FUNCTION_BLOCK CallButtons (* Composite Function Block Type *)
  (* Standard: 61499-2 *)
  (* Version 0.0, 11/8/2016, Dmitry, nxtControl GmbH, template *)
  PACKAGE Main;
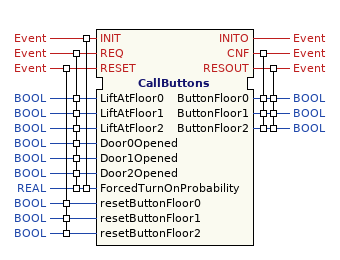
  EVENT_INPUT
    INIT WITH ForcedTurnOnProbability; (* Initialization Request *)
    REQ WITH LiftAtFloor0, LiftAtFloor1, LiftAtFloor2, Door0Opened, Door1Opened, Door2Opened, ForcedTurnOnProbability; (* Normal Execution Request *)
    RESET WITH resetButtonFloor0, resetButtonFloor1, resetButtonFloor2;
  END_EVENT
  EVENT_OUTPUT
    INITO; (* Initialization Confirm *)
    CNF WITH ButtonFloor0, ButtonFloor1, ButtonFloor2; (* Execution Confirmation *)
    RESOUT WITH ButtonFloor0, ButtonFloor1, ButtonFloor2;
  END_EVENT
  VAR_INPUT
    LiftAtFloor0 : BOOL; (* Input event qualifier *)
    LiftAtFloor1 : BOOL; (* Input event qualifier *)
    LiftAtFloor2 : BOOL; (* Input event qualifier *)
    Door0Opened : BOOL;
    Door1Opened : BOOL;
    Door2Opened : BOOL;
    ForcedTurnOnProbability : REAL;
    resetButtonFloor0 : BOOL;
    resetButtonFloor1 : BOOL;
    resetButtonFloor2 : BOOL;
  END_VAR
  VAR_OUTPUT
    ButtonFloor0 : BOOL; (* Output event qualifier *)
    ButtonFloor1 : BOOL; (* Output event qualifier *)
    ButtonFloor2 : BOOL; (* Output event qualifier *)
  END_VAR
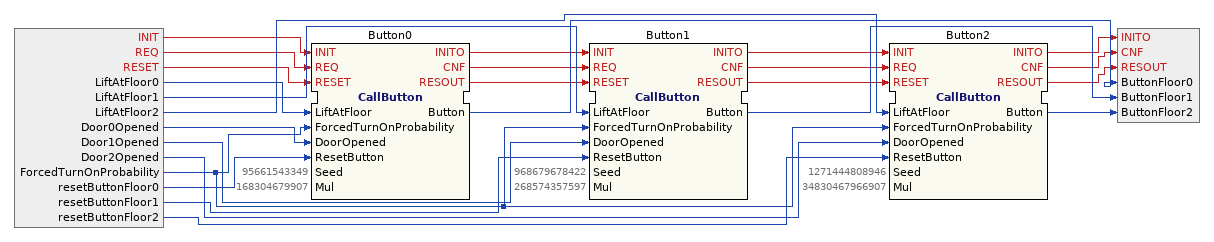
  FBS
    Button0 : CallButton(Seed := 95661543349, Mul := 168304679907);
    Button1 : CallButton(Seed := 968679678422, Mul := 268574357597);
    Button2 : CallButton(Seed := 1271444808946, Mul := 34830467966907);
  END_FBS
  EVENT_CONNECTIONS
    INIT TO Button0.INIT;
    REQ TO Button0.REQ;
    Button0.INITO TO Button1.INIT;
    Button1.INITO TO Button2.INIT;
    Button2.INITO TO INITO;
    Button0.CNF TO Button1.REQ;
    Button1.CNF TO Button2.REQ;
    Button2.CNF TO CNF;
    RESET TO Button0.RESET;
    Button0.RESOUT TO Button1.RESET;
    Button1.RESOUT TO Button2.RESET;
    Button2.RESOUT TO RESOUT;
  END_CONNECTIONS
  DATA_CONNECTIONS
    LiftAtFloor0 TO Button0.LiftAtFloor;
    LiftAtFloor1 TO Button1.LiftAtFloor;
    LiftAtFloor2 TO Button2.LiftAtFloor;
    ForcedTurnOnProbability TO Button0.ForcedTurnOnProbability;
    ForcedTurnOnProbability TO Button1.ForcedTurnOnProbability;
    ForcedTurnOnProbability TO Button2.ForcedTurnOnProbability;
    Door0Opened TO Button0.DoorOpened;
    Door1Opened TO Button1.DoorOpened;
    Door2Opened TO Button2.DoorOpened;
    Button0.Button TO ButtonFloor0;
    Button1.Button TO ButtonFloor1;
    Button2.Button TO ButtonFloor2;
    resetButtonFloor0 TO Button0.ResetButton;
    resetButtonFloor1 TO Button1.ResetButton;
    resetButtonFloor2 TO Button2.ResetButton;
  END_CONNECTIONS
END_FUNCTION_BLOCK
